(****************************************************************************************)
(*							Beckhoff Automation Poland									*)
(*								F_1stByteWtoB v1.0										*)
(*									15.02.2010											*)
(*		Funkcja wyciagajaca mniej znaczacy BYTE ze zmiennej typu WORD					*)
(*							 wyjscie typu BYTE											*)
(*______________________________________________________________________________________*)
FUNCTION F_1stByteWtoB : BYTE
VAR_INPUT
	wIn		:	WORD;
END_VAR

F_1stByteWtoB := WORD_TO_BYTE(wIn AND 16#FF);

END_FUNCTION

(* stored: Version 1.1.0.1, ProductVersion 3.1.4020.3
   POU F_1stByteWtoB: Id {373cc5ab-6125-4e27-b6b2-79fb5ccc3b33}, SpecialFunc None *)
